FUNCTION_BLOCK AnalogInput (* CAT Function Block Type *)
  (* Standard: 61499-2 *)
  (* Version 1.0, 10/7/2026, Claude/Hidryco, Schneider Electric, Rev1 - QualityFailDelay: tolerancia da falha de canal por qualidade do sinal (ChFailFilter + ChFailTimer); 0 = imediato, comportamento anterior. Alarmes BadQuality/UncertainQuality so com a falha confirmada. *)
  PACKAGE SE.Nereda;
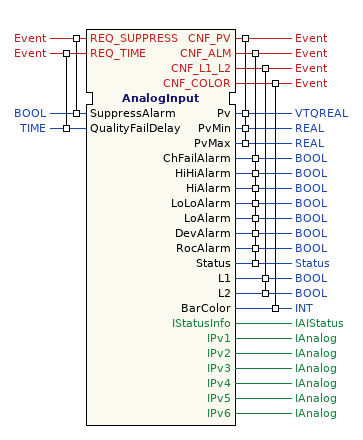
  EVENT_INPUT
    REQ_SUPPRESS WITH SuppressAlarm; (* Request to suppress the channel failure alarm *)
    REQ_TIME WITH QualityFailDelay;
  END_EVENT
  EVENT_OUTPUT
    CNF_PV WITH Pv, PvMin, PvMax; (* Execution confirmation of Pv *)
    CNF_ALM WITH ChFailAlarm, HiHiAlarm, HiAlarm, LoLoAlarm, LoAlarm, DevAlarm, RocAlarm, Status; (* Execution confirmation of alarm *)
    CNF_L1_L2 WITH L1, L2; (* Output Event *)
    CNF_COLOR WITH BarColor;
  END_EVENT
  VAR_INPUT
    SuppressAlarm : BOOL; (* 1 = Suppress channel failure in HMI *)
    QualityFailDelay : TIME := T#5s; (* Tolerancia da falha de canal por qualidade do sinal: so acusa se durar este tempo (0 = imediato, comportamento anterior) *)
  END_VAR
  VAR_OUTPUT
    Pv : VTQREAL; (* Scaled process signal *)
    PvMin : REAL; (* Minimum pv measurement range (in engineering units) *)
    PvMax : REAL; (* Maximun pv measurement range (in engineering units) *)
    ChFailAlarm : BOOL; (* 1 = Alarm condition is true with considering the suppress status *)
    HiHiAlarm : BOOL; (* 1 = high high alarm limit reached *)
    HiAlarm : BOOL; (* 1 = high alarm limit reached *)
    LoLoAlarm : BOOL; (* 1 = Low low alarm limit reached *)
    LoAlarm : BOOL; (* 1 = low Alarm limit reached *)
    DevAlarm : BOOL; (* 1 = Deviation alarm limit reached *)
    RocAlarm : BOOL; (* 1 = ROC alarm limit reached *)
    Status : Status; (* Status structure data (State alarm, HiHi alarm, Hi alarm, Lo alarm, LoLo alarm, Deviation alarm, Deviation Hi, Deivation Lo, ROC alarm, ROC Hi, ROC Lo, Min activated, Max activated) *)
    L1 : BOOL; (* Output event qualifier *)
    L2 : BOOL; (* Output event qualifier *)
    BarColor : INT;
  END_VAR
  PLUGS
    IStatusInfo : IAIStatus;
    IPv1 : IAnalog; (* Process value and status interface adapter *)
    IPv2 : IAnalog; (* Process value and status interface adapter *)
    IPv3 : IAnalog; (* Process value and status interface adapter *)
    IPv4 : IAnalog; (* Process value and status interface adapter *)
    IPv5 : IAnalog; (* Process value and status interface adapter *)
    IPv6 : IAnalog; (* Process value and status interface adapter *)
  END_PLUGS
  (* 01 - FUNCTIONNAL INPUT INTERFACE *)
  (* 00 - INITIALIZATION *)
  (* 05 - LOGIC *)
  (* 06 - HMI INTERFACE *)
  (* 04 - CHILDREN *)
  (* 03 - FIELD INTERFACE *)
  (* 02 - FUNCTIONNAL OUTPUT INTERFACE *)
  (* 07- Input Hardware Interface *)
  (* 4A - TYPICALS *)
  (* High high *)
  (* Deviation *)
  (* RateOfChange *)
  (* High *)
  (* Low *)
  (* Low Low *)
  (* Encode Status *)
  (* Encode Status *)
  (* L1 & L2 *)
  (* Channel Failure - Ovverride - Signal Quality *)
  (* 07- ±OTOR VS ALARM *)
  FBS
    AnalogInput : AnalogInputBase;
    rawPv : aISignal(Name := '$${PATH}AIn');
    StatusInfo : StatusInfo;
    IThis : AnalogInput_HMI(QI := TRUE);
    INIT : plcStart(Prio := 22, Delay := T#0ms);
    highHigh : LimitAlarm; {SET_ATTRIBUTE(HMI.AlarmText, $key:SE.App2CommonProcess.TxtHiHiLimit)} {SET_ATTRIBUTE(Configuration.Component.HideUnusedPorts, )}
    rateOfChange : ROCAlarm; {SET_ATTRIBUTE(HMI.AlarmText, $key:SE.App2CommonProcess.TxtRocLimit)} {SET_ATTRIBUTE(Configuration.Component.HideUnusedPorts, )}
    high : LimitAlarm; {SET_ATTRIBUTE(HMI.AlarmText, $key:SE.App2CommonProcess.TxtHiLimit)} {SET_ATTRIBUTE(Configuration.Component.HideUnusedPorts, )}
    low : LimitAlarm; {SET_ATTRIBUTE(HMI.AlarmText, $key:SE.App2CommonProcess.TxtLoLimit)} {SET_ATTRIBUTE(Configuration.Component.HideUnusedPorts, )}
    lowLow : LimitAlarm; {SET_ATTRIBUTE(HMI.AlarmText, $key:SE.App2CommonProcess.TxtLoLoLimit)} {SET_ATTRIBUTE(Configuration.Component.HideUnusedPorts, )}
    deviation : DeviationAlarm; {SET_ATTRIBUTE(HMI.AlarmText, $key:SE.App2CommonProcess.TxtDeviationLimit)} {SET_ATTRIBUTE(Configuration.Component.HideUnusedPorts, )}
    HighHighAnalog : encodeIAnalog; {SET_ATTRIBUTE(Configuration.Component.HideUnusedPorts, )}
    CNF_ALARM : E_MERGE_12;
    HighAnalog : encodeIAnalog; {SET_ATTRIBUTE(Configuration.Component.HideUnusedPorts, )}
    LowAnalog : encodeIAnalog; {SET_ATTRIBUTE(Configuration.Component.HideUnusedPorts, )}
    LowLowAnalog : encodeIAnalog; {SET_ATTRIBUTE(Configuration.Component.HideUnusedPorts, )}
    LowAnalog1 : encodeIAnalog; {SET_ATTRIBUTE(Configuration.Component.HideUnusedPorts, )}
    LowLowAnalog1 : encodeIAnalog; {SET_ATTRIBUTE(Configuration.Component.HideUnusedPorts, )}
    MultiAnalog : MultiAnalog;
    L1_Generator : LevelSetPoint(pin_E22497432101E9D3 := 0.01);
    L2_Generator : LevelSetPoint(pin_E22497432101E9D3 := 0.01);
    L1_Smmoth : boolValueChanged;
    L2_Smmoth : boolValueChanged;
    L1L2 : E_MERGE;
    PvStatus : AnalogStatus; {SET_ATTRIBUTE(Configuration.Component.HideUnusedPorts, )}
    SignalDecode : aiSignalDecode;
    ChFailure : OR_169B00D031196E7C4; {SET_ATTRIBUTE(Configuration.GenericFBType.InterfaceParams, Runtime.Standard#CNT:=4;OUT:BOOL)}
    ChFailureSmooth : boolValueChanged;
    FlowConvertUnit : ConvertFlowUnit;
    BadQuality : ALARM_BIT(ACKTYPE_1 := 2, ACTIVE := TRUE, TYPE := 1);
    UncertainQuality : ALARM_BIT(ACKTYPE_1 := 2, ACTIVE := TRUE, TYPE := 1);
    rawPvInt : SYMLINKMULTIVARDST_5A03F112CD5D470(QI := TRUE, NAME1 := '$${PATH}AInInt'); {SET_ATTRIBUTE(Configuration.GenericFBType.InterfaceParams, Runtime.System#I:=1;VALUE${I$}:INT)}
    rawPvIntConv : aiIntToVtqReal;
    ChFailFilter : QualityFailFilter;
    ChFailTimer : E_DELAY;
  END_FBS
  EVENT_CONNECTIONS
    L1L2.EO TO CNF_L1_L2;
    L1_Smmoth.CHD TO L1L2.EI1;
    L2_Smmoth.CHD TO L1L2.EI2;
    AnalogInput.CNF_PV TO HighHighAnalog.REQ;
    HighHighAnalog.CNF_FB TO PvStatus.F79B6341372EBAF9;
    AnalogInput.CNF_PV TO HighAnalog.REQ;
    HighAnalog.CNF_FB TO PvStatus.F79B6341372EBAF9;
    AnalogInput.CNF_PV TO LowAnalog.REQ;
    LowAnalog.CNF_FB TO PvStatus.F79B6341372EBAF9;
    AnalogInput.CNF_PV TO LowLowAnalog.REQ;
    LowLowAnalog.CNF_FB TO PvStatus.F79B6341372EBAF9;
    AnalogInput.CNF_PV TO LowAnalog1.REQ;
    LowAnalog1.CNF_FB TO PvStatus.F79B6341372EBAF9;
    deviation.CNF TO CNF_ALARM.EI5;
    AnalogInput.CNF_PV TO LowLowAnalog1.REQ;
    LowLowAnalog1.CNF_FB TO PvStatus.F79B6341372EBAF9;
    rateOfChange.CNF TO CNF_ALARM.EI6;
    AnalogInput.CNF_PV TO PvStatus.CC97B7AB29FD1036;
    highHigh.CNF TO CNF_ALARM.EI1;
    high.CNF TO CNF_ALARM.EI2;
    low.CNF TO CNF_ALARM.EI3;
    lowLow.CNF TO CNF_ALARM.EI4;
    CNF_ALARM.EO TO CNF_ALM;
    L1_Generator.5C15B34FA0BE2D12 TO L1_Smmoth.REQ;
    L2_Generator.5C15B34FA0BE2D12 TO L2_Smmoth.REQ;
    AnalogInput.CNF_PV TO L1_Generator.F1EF33EDF930102A;
    AnalogInput.CNF_PV TO L2_Generator.F1EF33EDF930102A;
    FlowConvertUnit.CNF TO AnalogInput.REQ_PV;
    REQ_SUPPRESS TO AnalogInput.REQ_SUPPRESS;
    AnalogInput.CNF_PV TO CNF_PV;
    PvStatus.C722264540EEA1B1 TO CNF_ALARM.61E483B0D1B23F8E;
    rawPv.CNF TO SignalDecode.4913BACAD6826E20;
    ChFailureSmooth.CHD TO PvStatus.F79B6341372EBAF9;
    ChFailureSmooth.CHD TO CNF_ALARM.523A3C57C3E4FA0F;
    ChFailureSmooth.CHD TO StatusInfo.7B1B2ACCEA05C392;
    AnalogInput.CNF_ALM TO ChFailure.REQ;
    FlowConvertUnit.CNF TO ChFailure.REQ;
    AnalogInput.CNF_PV TO ChFailure.REQ;
    AnalogInput.CNF_PV TO StatusInfo.E7A7AB00DEC6E3EC;
    SignalDecode.4B866291E3506649 TO FlowConvertUnit.REQ;
    BadQuality.INITO TO UncertainQuality.INIT;
    BadQuality.CNF_INITDATA TO BadQuality.REQ;
    BadQuality.CNF_INITDATA TO BadQuality.ACTIVATE;
    UncertainQuality.CNF_INITDATA TO UncertainQuality.ACTIVATE;
    UncertainQuality.CNF_INITDATA TO UncertainQuality.REQ;
    INIT.FIRST_INIT TO IThis.8605D25FEED5153E;
    INIT.REDO_INIT TO IThis.8605D25FEED5153E;
    L1L2.EO TO IThis.97DA89B5B690DDE2;
    AnalogInput.CNF_PV TO IThis.97DA89B5B690DDE2;
    highHigh.CNF_LIMITSP TO IThis.A2C25AD55AC2FADB;
    high.CNF_LIMITSP TO IThis.A2C25AD55AC2FADB;
    low.CNF_LIMITSP TO IThis.A2C25AD55AC2FADB;
    lowLow.CNF_LIMITSP TO IThis.A2C25AD55AC2FADB;
    highHigh.CNF TO IThis.A2C25AD55AC2FADB;
    high.CNF TO IThis.A2C25AD55AC2FADB;
    low.CNF TO IThis.A2C25AD55AC2FADB;
    lowLow.CNF TO IThis.A2C25AD55AC2FADB;
    highHigh.IND TO IThis.A2C25AD55AC2FADB;
    high.IND TO IThis.A2C25AD55AC2FADB;
    low.IND TO IThis.A2C25AD55AC2FADB;
    lowLow.IND TO IThis.A2C25AD55AC2FADB;
    IThis.3C13ABA26881DB90 TO IThis.E3E6A353D0B3EBA2;
    IThis.EB2BD10A2F1BC62E TO IThis.77446B0CC127CEA9;
    ChFailureSmooth.CHD TO IThis.267A885FF9BC7B84;
    IThis.81EC65B5ED359979 TO IThis.BDBFFF524FC5539D;
    IThis.81EC65B5ED359979 TO BadQuality.INIT;
    IThis.EB2BD10A2F1BC62E TO CNF_COLOR;
    IThis.CE82A4C836731358 TO L1_Generator.F1EF33EDF930102A;
    IThis.CE82A4C836731358 TO L2_Generator.F1EF33EDF930102A;
    IThis.E0AE911BEA30560A TO FlowConvertUnit.REQ;
    UncertainQuality.INITO TO INIT.ACK_FIRST;
    UncertainQuality.INITO TO BadQuality.REQ_INITDATA;
    UncertainQuality.INITO TO UncertainQuality.REQ_INITDATA;
    INIT.FIRST_INIT TO rawPvInt.INIT;
    INIT.REDO_INIT TO rawPvInt.INIT;
    rawPvInt.CNF TO rawPvIntConv.9C64D832256C82B4;
    rawPvIntConv.BC5EA87CD2275B61 TO SignalDecode.F08F00BBF3A56140;
    ChFailure.CNF TO ChFailFilter.D0DAEC8E3A7B0649;
    ChFailFilter.4A90895B1386766B TO ChFailureSmooth.REQ;
    ChFailFilter.4A90895B1386766B TO BadQuality.REQ;
    ChFailFilter.4A90895B1386766B TO UncertainQuality.REQ;
    ChFailFilter.9F58EC819BE28CD6 TO ChFailTimer.START;
    ChFailFilter.D03D083CB42919B5 TO ChFailTimer.STOP;
    ChFailTimer.EO TO ChFailFilter.5ACBE650D38A1821;
  END_CONNECTIONS
  DATA_CONNECTIONS
    highHigh.LimitReached TO HiHiAlarm;
    high.LimitReached TO HiAlarm;
    low.LimitReached TO LoAlarm;
    lowLow.LimitReached TO LoLoAlarm;
    rateOfChange.LimitReached TO RocAlarm;
    deviation.LimitReached TO DevAlarm;
    L1_Smmoth.Output TO L1;
    L2_Smmoth.Output TO L2;
    AnalogInput.Pv TO HighHighAnalog.Value;
    AnalogInput.PvMax TO HighHighAnalog.ValueHi;
    AnalogInput.PvMin TO HighHighAnalog.ValueLo;
    HighHighAnalog.Track TO PvStatus.28AAB407A0D794F9;
    AnalogInput.Pv TO HighAnalog.Value;
    AnalogInput.PvMax TO HighAnalog.ValueHi;
    AnalogInput.PvMin TO HighAnalog.ValueLo;
    HighAnalog.Track TO PvStatus.D77FE69E58404C72;
    AnalogInput.Pv TO LowAnalog.Value;
    AnalogInput.PvMax TO LowAnalog.ValueHi;
    AnalogInput.PvMin TO LowAnalog.ValueLo;
    LowAnalog.Track TO PvStatus.322FCCCFF0474AF4;
    LowLowAnalog.Track TO PvStatus.F7613467CAB82A70;
    AnalogInput.Pv TO LowLowAnalog.Value;
    AnalogInput.PvMax TO LowLowAnalog.ValueHi;
    AnalogInput.PvMin TO LowLowAnalog.ValueLo;
    LowAnalog1.Track TO PvStatus.C23A41885F1E1D50;
    AnalogInput.Pv TO LowAnalog1.Value;
    AnalogInput.PvMax TO LowAnalog1.ValueHi;
    AnalogInput.PvMin TO LowAnalog1.ValueLo;
    AnalogInput.Pv TO LowLowAnalog1.Value;
    AnalogInput.PvMax TO LowLowAnalog1.ValueHi;
    AnalogInput.PvMin TO LowLowAnalog1.ValueLo;
    LowLowAnalog1.Track TO PvStatus.450B11233AE13742;
    AnalogInput.Pv TO PvStatus.5D89DB5187B2462E;
    AnalogInput.PvMin TO PvStatus.7C99DC458353F065;
    AnalogInput.PvMax TO PvStatus.351FAAB35D0B0C22;
    L1_Generator.20BAB588313AD38F TO L1_Smmoth.Input;
    L2_Generator.20BAB588313AD38F TO L2_Smmoth.Input;
    AnalogInput.Pv TO L1_Generator.E7E7E59B5B35FDF5;
    AnalogInput.Pv TO L2_Generator.E7E7E59B5B35FDF5;
    FlowConvertUnit.OUT1 TO AnalogInput.RawPvIn;
    SuppressAlarm TO AnalogInput.SuppressAlarm;
    AnalogInput.Pv TO Pv;
    AnalogInput.PvMin TO PvMin;
    AnalogInput.PvMax TO PvMax;
    PvStatus.99E85C240FC6CE5E TO Status;
    ChFailureSmooth.Output TO PvStatus.E245520D1557B54B;
    ChFailureSmooth.Output TO ChFailAlarm;
    ChFailureSmooth.Output TO StatusInfo.934AEF6651857CA5;
    AnalogInput.ChFailAlarm TO ChFailure.IN1;
    SignalDecode.E756592F7CB68AC4 TO ChFailure.IN2;
    SignalDecode.201BC7AF68EF33E6 TO ChFailure.IN3;
    AnalogInput.BCEE37427EBF3A7A TO StatusInfo.669381E3EE065A76;
    SignalDecode.03C2FCFDEE2F946C TO FlowConvertUnit.IN1;
    AnalogInput.Pv TO IThis.593B0C1BA9886648;
    AnalogInput.PvMin TO IThis.E62EB46A29FA5F14;
    AnalogInput.PvMax TO IThis.793D93026D4B0479;
    L1_Smmoth.Output TO IThis.75726770057391E4;
    L2_Smmoth.Output TO IThis.1231178915ED30B5;
    highHigh.LimitSp TO IThis.89F139E97BA0A8F9;
    high.LimitSp TO IThis.D51D9F40AF5563F5;
    low.LimitSp TO IThis.B96DA755CCABAD3E;
    lowLow.LimitSp TO IThis.7D61380FB64EA01E;
    highHigh.Alarm TO IThis.443B6AA4B96CFD62;
    high.Alarm TO IThis.8D01629C22161E88;
    low.Alarm TO IThis.8006932B7C983E0F;
    lowLow.Alarm TO IThis.CB8A9984BB686A05;
    IThis.52DF787FBA5487DB TO IThis.411FEFE8AADAE8ED;
    IThis.45FE230A1EA15892 TO IThis.D835CDAA9E74318D;
    IThis.A311101D3C537B2D TO IThis.4209CA9DC93C4AA8;
    ChFailureSmooth.Output TO IThis.EC2E64A29E9C1CF2;
    AnalogInput.BCEE37427EBF3A7A TO IThis.621B1BF4799BDF6C;
    highHigh.Disabled TO IThis.622D95C981E27C66;
    high.Disabled TO IThis.33288C5A3BA1817F;
    low.Disabled TO IThis.2C2D5C1059052CF3;
    lowLow.Disabled TO IThis.5871750C82E7E712;
    IThis.A311101D3C537B2D TO BarColor;
    IThis.E76FE87B326922DA TO L1_Generator.B3F14A30A9C6E91C;
    IThis.BF5A04A4EC9A2DFE TO L2_Generator.B3F14A30A9C6E91C;
    IThis.12285BAA45AA2557 TO FlowConvertUnit.88326FC8282011A9;
    rawPv.Out TO SignalDecode.6969F2D522DDBD33;
    rawPvInt.VALUE1 TO rawPvIntConv.A7451C41429F9D06;
    rawPvInt.QO TO rawPvIntConv.9F9B5A9C85DA55C7;
    rawPvIntConv.6E40BF80683FA37C TO SignalDecode.D6314ADEFE23DADC;
    rawPvIntConv.FD829B78B964F3C2 TO SignalDecode.3126FE57F7AC4016;
    ChFailure.OUT TO ChFailFilter.BEF204F0906FF6D8;
    SignalDecode.E756592F7CB68AC4 TO ChFailFilter.47B2104419F3BB19;
    SignalDecode.201BC7AF68EF33E6 TO ChFailFilter.D0B962A0DD67BC30;
    QualityFailDelay TO ChFailFilter.802A68C220DBE1BD;
    ChFailFilter.D2C9F0958E4C098A TO ChFailureSmooth.Input;
    ChFailFilter.1A1043D3C0733A7D TO BadQuality.INP;
    ChFailFilter.1A6AD5B0D24F0EA5 TO UncertainQuality.INP;
    QualityFailDelay TO ChFailTimer.DT;
  END_CONNECTIONS
  ADAPTER_CONNECTIONS
    HighHighAnalog.IAnalog TO highHigh.IPv;
    HighAnalog.IAnalog TO high.IPv;
    LowAnalog.IAnalog TO low.IPv;
    LowLowAnalog.IAnalog TO lowLow.IPv;
    LowAnalog1.IAnalog TO deviation.IPv;
    LowLowAnalog1.IAnalog TO rateOfChange.IPv;
    PvStatus.D3137B5BC9BF5E62 TO MultiAnalog.8AE3BBA7BE7B68A3;
    MultiAnalog.3FB5E8550AE3652A TO IPv1;
    MultiAnalog.2B13B17B512405B9 TO IPv2;
    MultiAnalog.ABF3E5BD1080FA06 TO IPv3;
    MultiAnalog.2F696D2C94BC15F3 TO IPv4;
    MultiAnalog.0C612553273B91A4 TO IPv5;
    MultiAnalog.30DD549C419DF3C1 TO IPv6;
    StatusInfo.02A8A91DFB8F3CD3 TO IStatusInfo;
  END_CONNECTIONS
END_FUNCTION_BLOCK
